FUNCTION_BLOCK Heating_State_Heatup EXTENDS Heating_State
VAR_INPUT
END_VAR
VAR_OUTPUT
END_VAR
VAR
END_VAR

METHOD CanActivate : BOOL
CanActivate :=  _ctx.state.iMgr.Current = _ctx.state.iEnable;
END_METHOD

METHOD OnExecute
IF _ctx.hmi.bButton THEN
	_ctx.hmi.bButton := FALSE;
	_ctx.state.iMgr.Request(_ctx.state.iEnable);
END_IF
END_METHOD

METHOD OnInit
_ctx.hmi.sStatusText := 'Heating enabled: Heating up...';
_ctx.hmi.nStatusColor := COL.BLACK.Raw;

_ctx.hmi.sButtonText := 'Press to DISABLE!';
_ctx.hmi.nButtonColor := COL.BLACK.Raw;

_ctx.io.out.bBurner := TRUE;
_ctx.io.out.bPump := TRUE;
END_METHOD

END_FUNCTION_BLOCK

(* stored: Version 1.1.0.1
   POU Heating_State_Heatup: Id {7fc41e36-df57-4694-9616-ae401df4b5ef}, SpecialFunc None
   Method CanActivate: Id {f05d18ba-d846-47dc-8c6e-a43c0921ca66}
   Method OnExecute: Id {1e385c1c-ab42-445b-8b2a-c386ab10b6e6}
   Method OnInit: Id {625eecf1-2f5e-4832-964f-a20b5cc15fa9} *)
